PROGRAM main
  VAR
    LocalVar : DINT;
  END_VAR

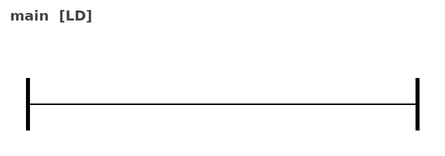
(* LD diagram, written out as Structured Text *)
END_PROGRAM
